{attribute 'GeneratedUsingTerminal: EL3773-0000-0018'}
{attribute addProperty BoxType "EL3773-0000-0018"}
{attribute addProperty Id "U2_SamplesAT %I*U2_Samples_2D13B74B20"}
{attribute addProperty CRC "2786968797"}
{attribute addProperty Size "20"}
TYPE L2_Voltage_Samples_A61DC4DD EXTENDS InputBase_8311D824 :
STRUCT
	{attribute addProperty Name "U2_Samples"}
	U2_Samples AT %I* : U2_Samples_2D13B74B;
END_STRUCT
END_TYPE

(* stored: Version 1.2.0.0, ProductVersion 3.1.4024.9
   DUT L2_Voltage_Samples_A61DC4DD: Id {2377017c-4d93-41c2-9d57-20e3a54388e2} *)
